// TIA Portal V17 export
// export: Created 2024-08-29T18:23:47.4399057Z, ExportSetting WithDefaults, DisplayName Totally Integrated Automation Portal, DisplayVersion V17 Update 7, DisplayName TIA Portal Openness, DisplayVersion V17 Update 7, DisplayName TIA Portal Version Control Interface, DisplayVersion V17, DisplayName SINAMICS Startdrive Advanced, DisplayVersion V17 SP2, DisplayName SINAMICS Startdrive G110M, G120, G120C, G120D, G120P, G115D, DisplayVersion V17 SP2, DisplayName SINAMICS Startdrive G130, G150, S120, S150, SINAMICS MV, S210, DisplayVersion V17 SP2, DisplayName STEP 7 Professional, DisplayVersion V17 Update 7, DisplayName STEP 7 Safety, DisplayVersion V17 Update 6, DisplayName WinCC Advanced / Unified PC, DisplayVersion V17 Update 7
DATA_BLOCK "timeSystemDB"   // DB32
VERSION : 0.1
// stored: AutoNumber true, DBAccessibleFromOPCUA true, DBAccessibleFromWebserver true, InstanceOfName timeSystem, InstanceOfType FB
"timeSystem"
   // VAR_INPUT
   //    bPartOkNok : Bool := FALSE;
   //    bRunningcycle : Bool := FALSE;
   //    bPreCount : Bool := FALSE;
   // END_VAR
   // VAR_OUTPUT
   //    bShift1 : Bool := FALSE;
   //    bShift2 : Bool := TRUE;
   //    bShift3 : Bool := FALSE;
   //    nCycle_Time_Shift : Real := 0.0;
   //    nCycleTimeAvg_Shift1 : Real := 0.0;
   //    nCycleTimeAvg_Shift2 : Real := 0.0;
   //    nCycleTimeAvg_Shift3 : Real := 0.0;
   // END_VAR
   // VAR
   //    Ret_Val_WR { ExternalAccessible := 'False'; ExternalVisible := 'False'; ExternalWritable := 'False'} : USInt := 0;
   //    Ret_Val_RD { ExternalAccessible := 'False'; ExternalVisible := 'False'; ExternalWritable := 'False'} : USInt := 0;
   //    DTL_Set_Time : DTL := DTL#2024-08-01-18:50:00;
   //    DTL_Read_Time : DTL := DTL#2024-08-02-15:53:42.527892088;
   //    TOD_Read : Time_Of_Day := TOD#15:53:42.527;
   //    Date_Read : Date := D#1990-01-01;
   //    bAceptButtonHmiP : Bool := FALSE;
   //    bAcept_buttonHMI : Bool := FALSE;
   //    nSet_minute : Int := 50;
   //    nSet_Hour : Int := 18;
   //    nSet_Day : Int := 1;
   //    nSet_Month : Int := 8;
   //    nSet_Year : Int := 2024;
   //    nCycleTimeArray : Array[0..5] of Real;
   //    tCycleTime { S7_SetPoint := 'True'} : IEC_TIMER;
   //    nCycleTimeET : UDInt := 0;
   //    tCycleTimeTotal : UDInt := 0;
   //    bPartOkNokP : Bool := FALSE;
   //    bPartOkNokCmd : Bool := FALSE;
   //    nPartAvgCounter : Int := 0;
   //    bCycle_StartedP : Bool := FALSE;
   //    bSH1 : Bool := FALSE;
   //    bSH2 : Bool := TRUE;
   //    bSH3 : Bool := FALSE;
   //    nCycle_Time : Real := 0.0;
   //    nCycleTimeAvg : Real := 0.0;
   //    Read_Local_Time : DTL := DTL#1970-01-01-00:00:00;
   //    Read_System_Time : DTL := DTL#2024-08-02-15:53:42.527876040;
   //    Time_HMI_Set : DTL := DTL#2024-08-01-18:50:00;
   //    RetVal1 : Word := 16#0000;
   //    Retval2 : Word := 16#0000;
   //    Retval3 : Word := 16#0000;
   //    n : Int := 0;
   //    timesCounter { S7_SetPoint := 'True'} : IEC_COUNTER;
   // END_VAR
   // VAR RETAIN
   //    tCycle_Running : Real := 0.0;
   // END_VAR
   // VAR
   //    nCycleAvg : DInt := 0;
   //    nCycleTime_Total : Time_Of_Day := TOD#00:00:00;
   //    ntimeRun_conv : UDInt := 0;
   // END_VAR
BEGIN
   nCycleTimeArray[0..5] := 0.0;
   tCycleTime.PT := T#0MS;
   tCycleTime.IN := FALSE;
   timesCounter.CU := FALSE;
   timesCounter.CD := FALSE;
   timesCounter.R := FALSE;
   timesCounter.LD := FALSE;
   timesCounter.QU := FALSE;
   timesCounter.QD := FALSE;
   timesCounter.PV := 5;
   timesCounter.CV := 0;
END_DATA_BLOCK
